PROGRAM P_Demo_FB_BARReadShadingObjectsList
VAR
    fb : FB_BARReadShadingObjectsList;                            // 被演示 FB 实例
    bStart_in : BOOL := FALSE;
    sDataFile_in : STRING := '';
    sLogFile_in : STRING := '';
    sNetId_in : STRING := '';
    arrShadingObject_io : ARRAY[1..iShadingObjects] OF ST_BARShadingObject ;
    bBusy_out : BOOL;
    bError_out : BOOL;
    udiErrorId_out : UDINT;
    uiAmountOfSetsRead_out : UINT;
END_VAR

// ============================================================================
// Tc2_HVAC.FB_BARReadShadingObjectsList 演示程序
// ============================================================================
// 场景：把本 FB 实例化到一个 PLC 程序里，每周期单次调用；按需要把 VAR_INPUT 与
//       VAR_IN_OUT 接到工程信号；VAR_OUTPUT 写入对应监视变量。
// 价值：使用本 FB 比手写状态机 / 控制算法节省大量代码；与 Tc2_HVAC 体系内其它 FB
//       直接对接，命名 / 持久化 / 模式仲裁等约定一致。具体语义见 FB_BARReadShadingObjectsList.md 主文档。
// 验证步骤：
//   1. 右键 PLC 项目下 POUs 文件夹 → Add → Existing Item → 选本 .TcPOU 文件
//   2. 引用 Tc2_HVAC（References → Add library）
//   3. 编译 → 登录 → 运行
//   4. 在线写各 *_in 输入信号触发 FB；在线 monitor *_out 引脚观察状态
// ============================================================================

fb(
    bStart := bStart_in,
    sDataFile := sDataFile_in,
    sLogFile := sLogFile_in,
    sNetId := sNetId_in,
    arrShadingObject := arrShadingObject_io,
    bBusy => bBusy_out,
    bError => bError_out,
    udiErrorId => udiErrorId_out,
    uiAmountOfSetsRead => uiAmountOfSetsRead_out
);

END_PROGRAM

(* stored: Version 1.1.0.1, ProductVersion 3.1.4024.5
   POU P_Demo_FB_BARReadShadingObjectsList: Id {d571a689-d030-5c16-9088-4ac658f7498f}, SpecialFunc None *)
